// TIA Portal V18 export
TYPE "SORTER_SPEED_STATE"
// stored: IsFailsafeCompliant true
   STRUCT
      "!!SPEED_STATE_REC.SORTER_{index}_STOPPED$$" : Bool;
      "!!SPEED_STATE_REC.SORTER_{index}_ENCODER_HEALTHY$$" : Bool;
   END_STRUCT;
END_TYPE
